PROGRAM P_CoatingProtections
VAR
    	fbStripProtXRTMR1 : FB_MirrorTwoCoatingProtection := (
            sDevName := 'XRTMR1',
            nUpperCoatingBoundary := 13300000,
            nUpperCoatingBitmask := 2#0000_0011_1111_1111,
            sUpperCoatingType := 'B4C',
            nLowerCoatingBoundary := 11800000,
            nLowerCoatingBitMask := 2#1111_1110_0000_0000,
            sLowerCoatingType := 'B4C/Ni');

    	fbStripProtMR2L0 : FB_MirrorTwoCoatingProtection := (
            sDevName := 'MR2L0',
            nUpperCoatingBoundary := 14300000,
            nUpperCoatingBitmask := 2#1111_1110_0000_0000,
            sUpperCoatingType := 'Ni',
            nLowerCoatingBoundary := 12800000,
            nLowerCoatingBitMask := 2#0000_0011_1111_1111,
            sLowerCoatingType := 'B4C');
END_VAR

fbStripProtXRTMR1(
    nCurrentEncoderCount := MAIN.nEncCntYupXRTM1,
    neVRange := PMPS.PMPS_GVL.stCurrentBeamParameters.neVRange,
    FFO := GVL_PMPS.g_FastFaultOutput1);

END_PROGRAM

(* stored: Version 1.1.0.1, ProductVersion 3.1.4022.18
   POU P_CoatingProtections: Id {3eac67bd-ceb1-46f6-9fb2-5e3c0612d4cd}, SpecialFunc None *)
